(* CoDeSys 2.3 export: VERSION.EXP *)

(* Data type in STRUCT *)
TYPE Version :
STRUCT
	major: SINT;
	minor: SINT;
	patch: SINT;
END_STRUCT
END_TYPE
